FUNCTION_BLOCK ModeControl IMPLEMENTS I_Mode
VAR
	{attribute 'hide'}
	_CurrentMode : DINT := 1;
END_VAR

METHOD ChangeMode
VAR_INPUT
	RequestedMode : DINT;
END_VAR
IF (RequestedMode >= 1) THEN
	_CurrentMode := RequestedMode;
ELSE
	Trace.LogMessage('Mode Controller', 'Requested Mode is not Defined');
END_IF
END_METHOD

{attribute 'monitoring' := 'call'}
PROPERTY CurrentMode : DINT
GET
CurrentMode := _CurrentMode;
END_GET
END_PROPERTY

END_FUNCTION_BLOCK

(* stored: Version 1.1.0.1, ProductVersion 3.1.4026.18
   POU ModeControl: Id {77561641-1ab8-44f5-99d4-37f3fb200a36}, SpecialFunc None
   Method ChangeMode: Id {0574cbb0-7576-4b63-88c2-180504acf2f9}
   Property CurrentMode: Id {8ea7f208-a1f6-4963-8d0d-b4d4f4e4dd44}
   Get Get: Id {53ce988f-40e7-4999-91d1-9c988e1c2051} *)
